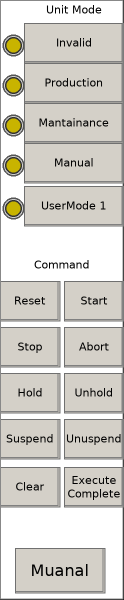
VISUALIZATION VIS_TemplateCommand  // 124x600
VAR_IN_OUT
	eModeCommand	: DINT;
	eStateCommand	: DINT;
	eModeStatus		: DINT;
	eStateStatus	: DINT;
	bModeChangeReq	: BOOL;
END_VAR
    Rectangle (0,0 124x600)
    Lamp1 (1,33 25x25), variable: (eModeStatus = 0), style: Lamp-Lamp1-Yellow
    Button (24,23 100x40), "Invalid", colour toggle: (eModeStatus = 0)
        tap bModeChangeReq
        OnMouseClick: execute { eModeCommand := 0; }
    Lamp1 (1,73 25x25), variable: (eModeStatus = 1), style: Lamp-Lamp1-Yellow
    Button (24,63 100x40), "Production"
        tap bModeChangeReq
        OnMouseClick: execute { eModeCommand := 1; }
    Lamp1 (1,113 25x25), variable: (eModeStatus = 2), style: Lamp-Lamp1-Yellow
    Button (24,103 100x40), "Mantainance"
        tap bModeChangeReq
        OnMouseClick: execute { eModeCommand := 2; }
    Lamp1 (1,153 25x25), variable: (eModeStatus = 3), style: Lamp-Lamp1-Yellow
    Button (24,143 100x40), "Manual"
        tap bModeChangeReq
        OnMouseClick: execute { eModeCommand := 3; }
    Lamp1 (1,196 25x25), variable: (eModeStatus = 4), style: Lamp-Lamp1-Yellow
    Button (24,186 100x40), "UserMode 1"
        tap bModeChangeReq
        OnMouseClick: execute { eModeCommand := 4; }
    Button (0,281 60x40), "Reset"
        OnMouseClick: execute { eStateCommand := 1; }
    Button (64,281 60x40), "Start"
        OnMouseClick: execute { eStateCommand := 2; }
    Button (0,327 60x40), "Stop"
        OnMouseClick: execute { eStateCommand := 3; }
    Button (0,373 60x40), "Hold"
        OnMouseClick: execute { eStateCommand := 4; }
    Button (64,373 60x40), "Unhold"
        OnMouseClick: execute { eStateCommand := 5; }
    Button (0,419 60x40), "Suspend"
        OnMouseClick: execute { eStateCommand := 6; }
    Button (64,419 60x40), "Unuspend"
        OnMouseClick: execute { eStateCommand := 7; }
    Button (0,467 60x40), "Clear"
        OnMouseClick: execute { eStateCommand := 9; }
    Label (0,255 124x20), "Command"
    Button (64,327 60x40), "Abort"
        OnMouseClick: execute { eStateCommand := 8; }
    Button (64,467 60x40), "Execute Complete"
        OnMouseClick: execute { MAIN.bExecuteComplete := TRUE; }
    Label (24,0 100x20), "Unit Mode"
    Button (15,548 90x45), "Muanal"
        p573394764: 16#FF000000 OR ( 16#FF00FF00)
        OnMouseDown: execute {
            IF G_HMI.iPML_mainFrame	= 0 THEN
            	G_HMI.iPML_mainFrame	:= 1;
            ELSE
            	G_HMI.iPML_mainFrame	:= 0;
            END_IF
        }
END_VISUALIZATION

(* stored: Version 1.1.0.1, ProductVersion 3.1.4024.12
   Visu VIS_TemplateCommand: Id {d7925750-20c5-4482-a15b-9b1c5b9b40e3} *)
